PROGRAM MAIN
VAR
	bteste: BOOL;
	iVar: INT := 0;
END_VAR

bteste;


//kkkk
iVar:=iVar+1;

END_PROGRAM

(* stored: Version 1.1.0.1, ProductVersion 3.1.4024.12
   POU MAIN: Id {da3c8636-7c7d-4b5a-ae28-b2fb9b62cf92}, SpecialFunc None *)
